PROGRAM sub_Security
VAR

END_VAR

//###################################################################################
//##-----------------------------------SECURITY------------------------------------##
//###################################################################################

//--------------------Variablen Setzen----------------------------------
//ALARM GESAMT
IF gvl_mb.Output_Coils[240] THEN
	gvl_mb.Output_Coils[241] 	:= TRUE;
	gvl_mb.Output_Coils[244]	:= TRUE;
END_IF

//ALARM LICHT
IF gvl_mb.Output_Coils[241] THEN
	gvl_mb.Output_Coils[242]	:= TRUE;
	gvl_mb.Output_Coils[243]	:= TRUE;
END_IF

//ALARM NOIS
IF gvl_mb.Output_Coils[244] THEN
	gvl_mb.Output_Coils[245]	:= TRUE;
	gvl_mb.Output_Coils[246]	:= TRUE;
END_IF


//--------------------------------- INVERT Input Windows / Doors ------------------------
gvl_mb.Output_Coils[200] := NOT gvl_EA.bID24_01_3;		// Fensterkontakt Bad EG
gvl_mb.Output_Coils[201] := NOT gvl_EA.bID24_01_4;		// Fensterkontakt Büro
gvl_mb.Output_Coils[203] := NOT gvl_EA.bID24_02_1;		// Fensterkontakt Keller
gvl_mb.Output_Coils[204] := NOT gvl_EA.bID24_02_2;		// Fensterkontakt Technik
gvl_mb.Output_Coils[205] := NOT gvl_EA.bID24_02_3;		// Fensterkontakt Hobbyraum Süd
gvl_mb.Output_Coils[207] := NOT gvl_EA.bID24_02_4;		// Kontakt Terassentür UG
gvl_mb.Output_Coils[206] := NOT gvl_EA.bID24_03_1;		// Fensterkontakt Hobbyraum West
gvl_mb.Output_Coils[202] := NOT gvl_EA.bID24_03_2;		// Kontakt Balkontür
gvl_mb.Output_Coils[209] := NOT gvl_EA.bWID01_3;		// Reedkontakt Werkstatttür
gvl_mb.Output_Coils[208] := NOT gvl_EA.bWID01_4;		// Reedkontakt Werkstattfenster
gvl_mb.Output_coils[210] :=	NOT gvl_EA.bWID01_11; 		// TüR		OG	Garage Strasse
gvl_mb.Output_coils[211] :=	NOT gvl_EA.bWID01_12; 		// Fenster	OG	Garage
gvl_mb.Output_Coils[212] :=	NOT gvl_EA.bWID01_13; 		// TüR		OG	Garage Haus

gvl_mb.Output_coils[213] :=	gvl_EA.bWID01_15; 			// Garagentor offen
gvl_mb.Output_coils[214] := gvl_EA.bWID01_16; 			// Garagentor geschlossen
gvl_mb.Output_Coils[215] := gvl_EA.bWID01_14; 			// Garagentor Lüftung

END_PROGRAM

(* stored: Version 1.1.0.1, ProductVersion 3.1.4024.4
   POU sub_Security: Id {cc922faa-17ab-4d35-9cbc-7ff8e2c57d1e}, SpecialFunc None *)
